REGION Network 69: Step [1291] : JOB[12] Step End
   RUNG wire#powerrail
      { S7_Templates := "SrcType := DInt" } EQ_Contact(in1 := "Unit1.Em7.ControlNodes".conveyor.sequence.status.currentStep, in2 := #JOB_12_STEP_91)
      Contact( "Unit1.Em7.ControlNodes".conveyor.sequence.status.seqActive )
      wire#w1
      Coil( "Unit1.Em7.ControlNodes".conveyor."step".action[1291] )
   END_RUNG
   RUNG wire#w1
      Coil( "Unit1.Em7.ControlNodes".conveyor."step".transition[1291] )
   END_RUNG
   RUNG wire#w1
      Contact( "Unit1.Em7.ControlNodes".conveyor."step".transition[1291] )
      { S7_Templates := "time_type := Time" } #statTonTimer[1291].TON(pt := #SeqNoDelayTime, et =>)
      Move(in := #STEP_IDLE, out1 => "Unit1.Em7.ControlNodes".conveyor.sequence.status.nextStep)
   END_RUNG
   // the same network as SCL:
   "Unit1.Em7.ControlNodes".conveyor."step".action[1291] := ("Unit1.Em7.ControlNodes".conveyor.sequence.status.currentStep = #JOB_12_STEP_91) AND "Unit1.Em7.ControlNodes".conveyor.sequence.status.seqActive;
   "Unit1.Em7.ControlNodes".conveyor."step".transition[1291] := ("Unit1.Em7.ControlNodes".conveyor.sequence.status.currentStep = #JOB_12_STEP_91) AND "Unit1.Em7.ControlNodes".conveyor.sequence.status.seqActive;
   #statTonTimer[1291].TON(IN := ("Unit1.Em7.ControlNodes".conveyor.sequence.status.currentStep = #JOB_12_STEP_91) AND "Unit1.Em7.ControlNodes".conveyor.sequence.status.seqActive AND "Unit1.Em7.ControlNodes".conveyor."step".transition[1291],
                           PT := #SeqNoDelayTime);
   IF #statTonTimer[1291].Q THEN
       "Unit1.Em7.ControlNodes".conveyor.sequence.status.nextStep := #STEP_IDLE;
   END_IF;
END_REGION

REGION Network 70: *************** IMMEDIATE STOP ****************
END_REGION

REGION Network 71: Immediate Stop
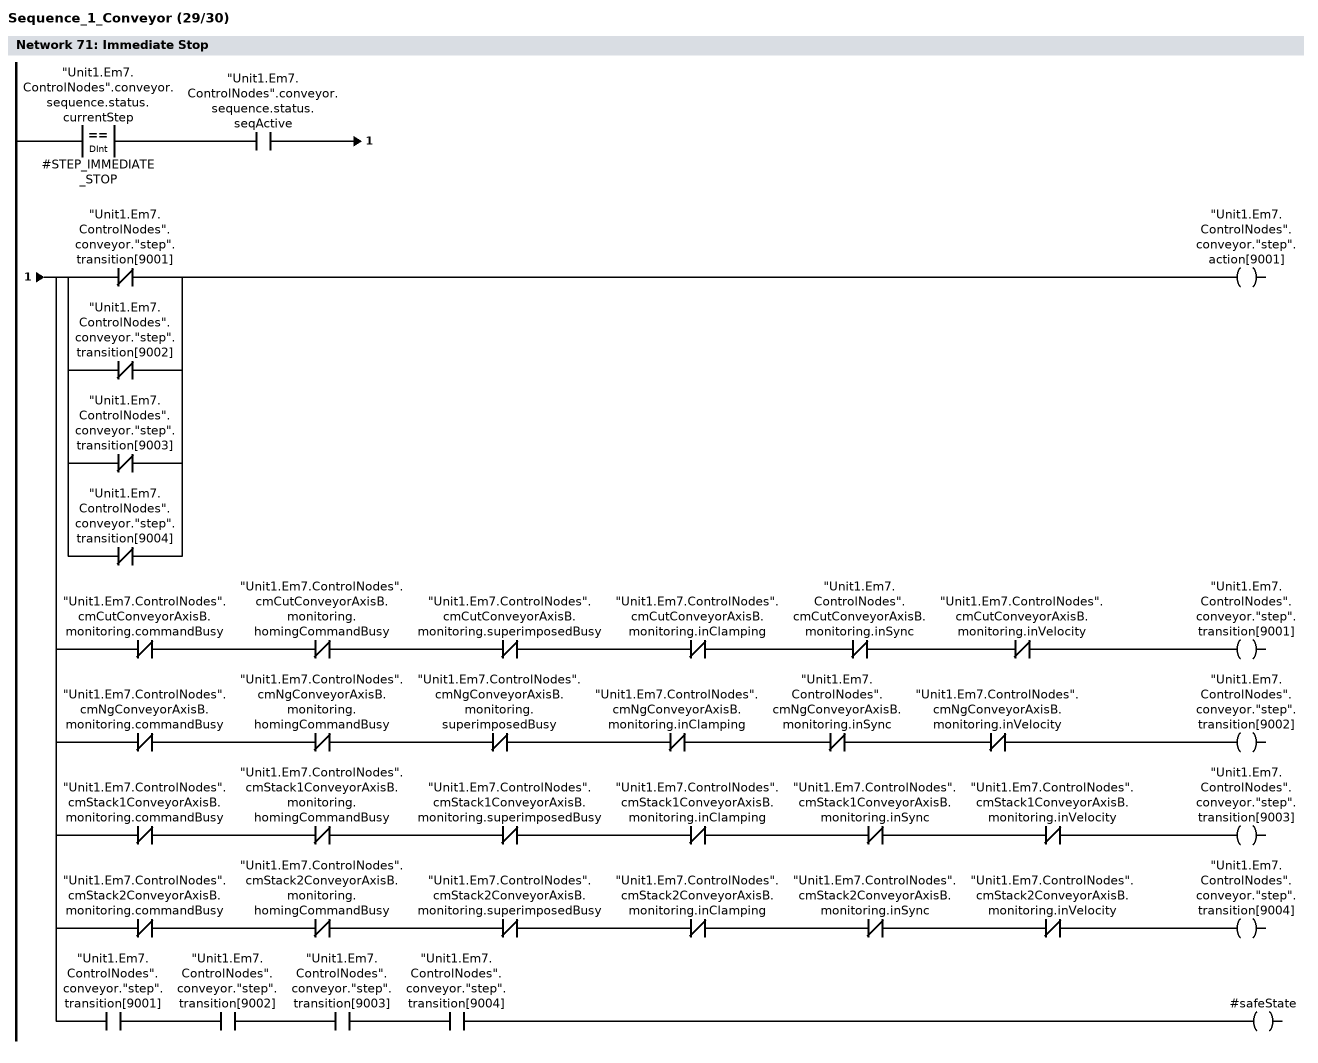
   RUNG wire#powerrail
      { S7_Templates := "SrcType := DInt" } EQ_Contact(in1 := "Unit1.Em7.ControlNodes".conveyor.sequence.status.currentStep, in2 := #STEP_IMMEDIATE_STOP)
      Contact( "Unit1.Em7.ControlNodes".conveyor.sequence.status.seqActive )
      wire#w1
      I_Contact( "Unit1.Em7.ControlNodes".conveyor."step".transition[9001] )
      wire#w2
      Coil( "Unit1.Em7.ControlNodes".conveyor."step".action[9001] )
   END_RUNG
   RUNG wire#w1
      I_Contact( "Unit1.Em7.ControlNodes".conveyor."step".transition[9002] )
   END_RUNG wire#w2
   RUNG wire#w1
      I_Contact( "Unit1.Em7.ControlNodes".conveyor."step".transition[9003] )
   END_RUNG wire#w2
   RUNG wire#w1
      I_Contact( "Unit1.Em7.ControlNodes".conveyor."step".transition[9004] )
   END_RUNG wire#w2
   RUNG wire#w1
      I_Contact( "Unit1.Em7.ControlNodes".cmCutConveyorAxisB.monitoring.commandBusy )
      I_Contact( "Unit1.Em7.ControlNodes".cmCutConveyorAxisB.monitoring.homingCommandBusy )
      I_Contact( "Unit1.Em7.ControlNodes".cmCutConveyorAxisB.monitoring.superimposedBusy )
      I_Contact( "Unit1.Em7.ControlNodes".cmCutConveyorAxisB.monitoring.inClamping )
      I_Contact( "Unit1.Em7.ControlNodes".cmCutConveyorAxisB.monitoring.inSync )
      I_Contact( "Unit1.Em7.ControlNodes".cmCutConveyorAxisB.monitoring.inVelocity )
      Coil( "Unit1.Em7.ControlNodes".conveyor."step".transition[9001] )
   END_RUNG
   RUNG wire#w1
      I_Contact( "Unit1.Em7.ControlNodes".cmNgConveyorAxisB.monitoring.commandBusy )
      I_Contact( "Unit1.Em7.ControlNodes".cmNgConveyorAxisB.monitoring.homingCommandBusy )
      I_Contact( "Unit1.Em7.ControlNodes".cmNgConveyorAxisB.monitoring.superimposedBusy )
      I_Contact( "Unit1.Em7.ControlNodes".cmNgConveyorAxisB.monitoring.inClamping )
      I_Contact( "Unit1.Em7.ControlNodes".cmNgConveyorAxisB.monitoring.inSync )
      I_Contact( "Unit1.Em7.ControlNodes".cmNgConveyorAxisB.monitoring.inVelocity )
      Coil( "Unit1.Em7.ControlNodes".conveyor."step".transition[9002] )
   END_RUNG
   RUNG wire#w1
      I_Contact( "Unit1.Em7.ControlNodes".cmStack1ConveyorAxisB.monitoring.commandBusy )
      I_Contact( "Unit1.Em7.ControlNodes".cmStack1ConveyorAxisB.monitoring.homingCommandBusy )
      I_Contact( "Unit1.Em7.ControlNodes".cmStack1ConveyorAxisB.monitoring.superimposedBusy )
      I_Contact( "Unit1.Em7.ControlNodes".cmStack1ConveyorAxisB.monitoring.inClamping )
      I_Contact( "Unit1.Em7.ControlNodes".cmStack1ConveyorAxisB.monitoring.inSync )
      I_Contact( "Unit1.Em7.ControlNodes".cmStack1ConveyorAxisB.monitoring.inVelocity )
      Coil( "Unit1.Em7.ControlNodes".conveyor."step".transition[9003] )
   END_RUNG
   RUNG wire#w1
      I_Contact( "Unit1.Em7.ControlNodes".cmStack2ConveyorAxisB.monitoring.commandBusy )
      I_Contact( "Unit1.Em7.ControlNodes".cmStack2ConveyorAxisB.monitoring.homingCommandBusy )
      I_Contact( "Unit1.Em7.ControlNodes".cmStack2ConveyorAxisB.monitoring.superimposedBusy )
      I_Contact( "Unit1.Em7.ControlNodes".cmStack2ConveyorAxisB.monitoring.inClamping )
      I_Contact( "Unit1.Em7.ControlNodes".cmStack2ConveyorAxisB.monitoring.inSync )
      I_Contact( "Unit1.Em7.ControlNodes".cmStack2ConveyorAxisB.monitoring.inVelocity )
      Coil( "Unit1.Em7.ControlNodes".conveyor."step".transition[9004] )
   END_RUNG
   RUNG wire#w1
      Contact( "Unit1.Em7.ControlNodes".conveyor."step".transition[9001] )
      Contact( "Unit1.Em7.ControlNodes".conveyor."step".transition[9002] )
      Contact( "Unit1.Em7.ControlNodes".conveyor."step".transition[9003] )
      Contact( "Unit1.Em7.ControlNodes".conveyor."step".transition[9004] )
      Coil( #safeState )
   END_RUNG
   // the same network as SCL:
   #_w1 := ("Unit1.Em7.ControlNodes".conveyor.sequence.status.currentStep = #STEP_IMMEDIATE_STOP) AND "Unit1.Em7.ControlNodes".conveyor.sequence.status.seqActive;
   "Unit1.Em7.ControlNodes".conveyor."step".action[9001] := #_w1 AND (NOT "Unit1.Em7.ControlNodes".conveyor."step".transition[9001] OR NOT "Unit1.Em7.ControlNodes".conveyor."step".transition[9002] OR NOT "Unit1.Em7.ControlNodes".conveyor."step".transition[9003] OR NOT "Unit1.Em7.ControlNodes".conveyor."step".transition[9004]);
   "Unit1.Em7.ControlNodes".conveyor."step".transition[9001] := #_w1 AND NOT "Unit1.Em7.ControlNodes".cmCutConveyorAxisB.monitoring.commandBusy AND NOT "Unit1.Em7.ControlNodes".cmCutConveyorAxisB.monitoring.homingCommandBusy AND NOT "Unit1.Em7.ControlNodes".cmCutConveyorAxisB.monitoring.superimposedBusy AND NOT "Unit1.Em7.ControlNodes".cmCutConveyorAxisB.monitoring.inClamping AND NOT "Unit1.Em7.ControlNodes".cmCutConveyorAxisB.monitoring.inSync AND NOT "Unit1.Em7.ControlNodes".cmCutConveyorAxisB.monitoring.inVelocity;
   "Unit1.Em7.ControlNodes".conveyor."step".transition[9002] := #_w1 AND NOT "Unit1.Em7.ControlNodes".cmNgConveyorAxisB.monitoring.commandBusy AND NOT "Unit1.Em7.ControlNodes".cmNgConveyorAxisB.monitoring.homingCommandBusy AND NOT "Unit1.Em7.ControlNodes".cmNgConveyorAxisB.monitoring.superimposedBusy AND NOT "Unit1.Em7.ControlNodes".cmNgConveyorAxisB.monitoring.inClamping AND NOT "Unit1.Em7.ControlNodes".cmNgConveyorAxisB.monitoring.inSync AND NOT "Unit1.Em7.ControlNodes".cmNgConveyorAxisB.monitoring.inVelocity;
   "Unit1.Em7.ControlNodes".conveyor."step".transition[9003] := #_w1 AND NOT "Unit1.Em7.ControlNodes".cmStack1ConveyorAxisB.monitoring.commandBusy AND NOT "Unit1.Em7.ControlNodes".cmStack1ConveyorAxisB.monitoring.homingCommandBusy AND NOT "Unit1.Em7.ControlNodes".cmStack1ConveyorAxisB.monitoring.superimposedBusy AND NOT "Unit1.Em7.ControlNodes".cmStack1ConveyorAxisB.monitoring.inClamping AND NOT "Unit1.Em7.ControlNodes".cmStack1ConveyorAxisB.monitoring.inSync AND NOT "Unit1.Em7.ControlNodes".cmStack1ConveyorAxisB.monitoring.inVelocity;
   "Unit1.Em7.ControlNodes".conveyor."step".transition[9004] := #_w1 AND NOT "Unit1.Em7.ControlNodes".cmStack2ConveyorAxisB.monitoring.commandBusy AND NOT "Unit1.Em7.ControlNodes".cmStack2ConveyorAxisB.monitoring.homingCommandBusy AND NOT "Unit1.Em7.ControlNodes".cmStack2ConveyorAxisB.monitoring.superimposedBusy AND NOT "Unit1.Em7.ControlNodes".cmStack2ConveyorAxisB.monitoring.inClamping AND NOT "Unit1.Em7.ControlNodes".cmStack2ConveyorAxisB.monitoring.inSync AND NOT "Unit1.Em7.ControlNodes".cmStack2ConveyorAxisB.monitoring.inVelocity;
   #safeState := #_w1 AND "Unit1.Em7.ControlNodes".conveyor."step".transition[9001] AND "Unit1.Em7.ControlNodes".conveyor."step".transition[9002] AND "Unit1.Em7.ControlNodes".conveyor."step".transition[9003] AND "Unit1.Em7.ControlNodes".conveyor."step".transition[9004];
END_REGION

REGION Network 72: *************** STATUS **********************
END_REGION

REGION Network 73: Sequence Status
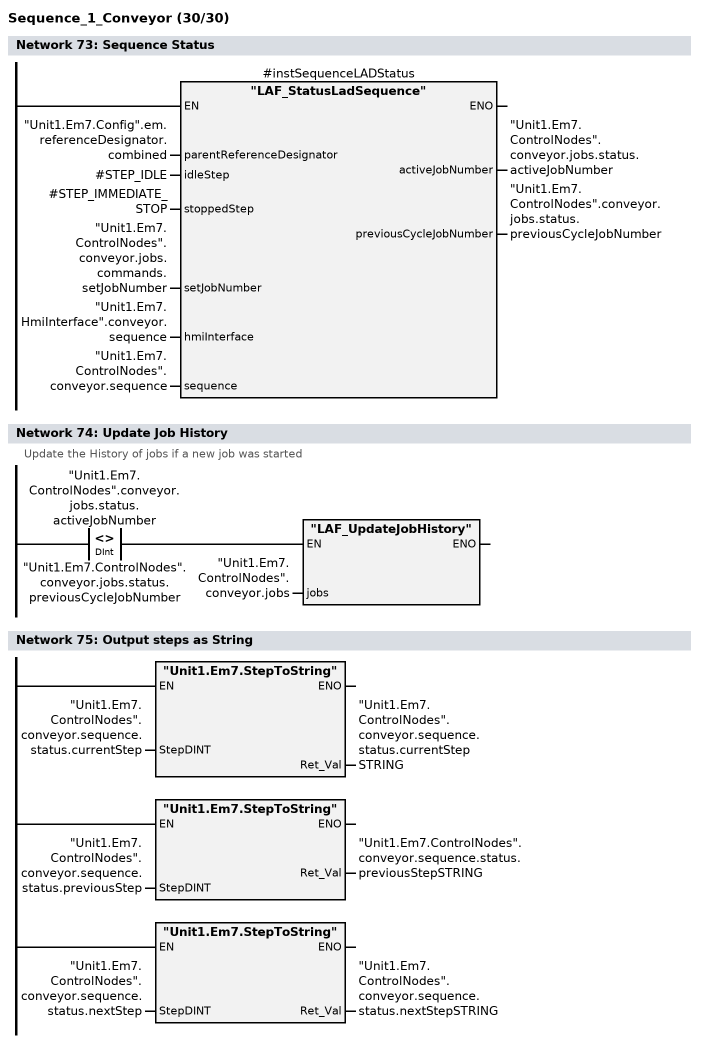
   RUNG wire#powerrail
      #instSequenceLADStatus(parentReferenceDesignator := "Unit1.Em7.Config".em.referenceDesignator.combined, idleStep := #STEP_IDLE, stoppedStep := #STEP_IMMEDIATE_STOP, setJobNumber := "Unit1.Em7.ControlNodes".conveyor.jobs.commands.setJobNumber, hmiInterface := "Unit1.Em7.HmiInterface".conveyor.sequence, sequence := "Unit1.Em7.ControlNodes".conveyor.sequence, activeJobNumber => "Unit1.Em7.ControlNodes".conveyor.jobs.status.activeJobNumber, previousCycleJobNumber => "Unit1.Em7.ControlNodes".conveyor.jobs.status.previousCycleJobNumber)
   END_RUNG
   // the same network as SCL:
   #instSequenceLADStatus(parentReferenceDesignator := "Unit1.Em7.Config".em.referenceDesignator.combined,   // "LAF_StatusLadSequence"
                          idleStep := #STEP_IDLE,
                          stoppedStep := #STEP_IMMEDIATE_STOP,
                          setJobNumber := "Unit1.Em7.ControlNodes".conveyor.jobs.commands.setJobNumber,
                          hmiInterface := "Unit1.Em7.HmiInterface".conveyor.sequence,
                          sequence := "Unit1.Em7.ControlNodes".conveyor.sequence,
                          activeJobNumber => "Unit1.Em7.ControlNodes".conveyor.jobs.status.activeJobNumber,
                          previousCycleJobNumber => "Unit1.Em7.ControlNodes".conveyor.jobs.status.previousCycleJobNumber);
END_REGION

REGION Network 74: Update Job History
   // Update the History of jobs if a new job was started
   RUNG wire#powerrail
      { S7_Templates := "SrcType := DInt" } NE_Contact(in1 := "Unit1.Em7.ControlNodes".conveyor.jobs.status.activeJobNumber, in2 := "Unit1.Em7.ControlNodes".conveyor.jobs.status.previousCycleJobNumber)
      "LAF_UpdateJobHistory"(jobs := "Unit1.Em7.ControlNodes".conveyor.jobs)
   END_RUNG
   // the same network as SCL:
   IF "Unit1.Em7.ControlNodes".conveyor.jobs.status.activeJobNumber <> "Unit1.Em7.ControlNodes".conveyor.jobs.status.previousCycleJobNumber THEN
       "LAF_UpdateJobHistory"(jobs := "Unit1.Em7.ControlNodes".conveyor.jobs);
   END_IF;
END_REGION

REGION Network 75: Output steps as String
   RUNG wire#powerrail
      "Unit1.Em7.StepToString"(StepDINT := "Unit1.Em7.ControlNodes".conveyor.sequence.status.currentStep, Ret_Val => "Unit1.Em7.ControlNodes".conveyor.sequence.status.currentStepSTRING)
   END_RUNG
   RUNG wire#powerrail
      "Unit1.Em7.StepToString"(StepDINT := "Unit1.Em7.ControlNodes".conveyor.sequence.status.previousStep, Ret_Val => "Unit1.Em7.ControlNodes".conveyor.sequence.status.previousStepSTRING)
   END_RUNG
   RUNG wire#powerrail
      "Unit1.Em7.StepToString"(StepDINT := "Unit1.Em7.ControlNodes".conveyor.sequence.status.nextStep, Ret_Val => "Unit1.Em7.ControlNodes".conveyor.sequence.status.nextStepSTRING)
   END_RUNG
   // the same network as SCL:
   "Unit1.Em7.ControlNodes".conveyor.sequence.status.currentStepSTRING := "Unit1.Em7.StepToString"(StepDINT := "Unit1.Em7.ControlNodes".conveyor.sequence.status.currentStep);
   "Unit1.Em7.ControlNodes".conveyor.sequence.status.previousStepSTRING := "Unit1.Em7.StepToString"(StepDINT := "Unit1.Em7.ControlNodes".conveyor.sequence.status.previousStep);
   "Unit1.Em7.ControlNodes".conveyor.sequence.status.nextStepSTRING := "Unit1.Em7.StepToString"(StepDINT := "Unit1.Em7.ControlNodes".conveyor.sequence.status.nextStep);
END_REGION
END_FUNCTION_BLOCK
